Yaskawa INFORM job: R1_72,2(0,0)R2.JBI

/JOB
//NAME R1_72,2(0,0)R2
///FOLDERNAME KRIS-SCIANA
//POS
///NPOS 57,57,0,3,0,0
///TOOL 0
///POSTYPE PULSE
///PULSE
C00000=120729,38464,-23607,67702,92694,37114
C00001=130813,19897,-28859,40674,87554,31415
C00002=125083,56704,30738,54224,74995,24956
C00003=126358,57000,31561,53980,74051,25086
C00004=124721,62288,44734,63185,73473,22335
C00005=124721,62512,45919,63338,73183,22075
C00006=124721,62288,44734,63185,73473,22335
C00007=125305,62416,44881,63099,73087,22421
C00008=124721,62288,44734,63185,73473,22335
C00009=120729,38464,-23607,67702,92694,37114
C00010=120728,81583,44137,67576,84483,28591
C00011=120728,81849,43244,67535,84761,28882
C00012=120728,81417,45180,67625,84187,28282
C00013=120728,81508,44709,67602,84324,28425
C00014=119180,81573,44789,67929,85318,28213
C00015=119180,81465,45362,67951,85156,28039
C00016=120171,81410,45292,67747,84521,28174
C00017=118840,81840,43784,67968,85844,28487
C00018=118840,81840,43784,67968,85844,28487
C00019=120728,81522,44639,67599,84344,28446
C00020=120728,81598,44155,67576,84481,28590
C00021=121739,82345,42246,50477,71891,30249
C00022=121737,83430,44678,50707,71287,29904
C00023=121727,86673,48704,50914,70767,29601
C00024=120728,82318,42212,50838,72434,30029
C00025=120728,82318,42212,50838,72434,30029
C00026=120728,83470,39162,50303,74040,30931
C00027=120731,108704,30437,520,103146,-53106
C00028=120730,95364,30685,507,96140,-53135
C00029=120729,92856,31465,505,94371,-53142
C00030=120882,90601,30856,459,93584,-53097
C00031=120076,91948,31897,698,93643,-53342
C00032=120729,92386,31163,506,94315,-53143
C00033=120916,97871,39788,450,91825,-53093
C00034=121066,129805,79437,461,95361,-53027
C00035=121134,131914,82339,451,94657,-53008
C00036=120821,132587,79324,499,96860,-53101
C00037=120730,97149,30254,16854,109142,-86058
C00038=94374,59905,-24624,-6692,95808,-73268
C00039=94859,43835,-17383,-4554,74801,-71238
C00040=94859,41415,-16000,-4599,72712,-71159
C00041=88285,47191,-10324,7479,76594,-70277
C00042=94590,38531,-17304,-4457,72022,-71215
C00043=94826,41033,-16151,-4582,72608,-71165
C00044=88838,46898,-10539,7187,76531,-70115
C00045=90938,44895,-12618,6065,76637,-69484
C00046=101911,56037,-3137,-16386,82833,-70668
C00047=102467,62438,3678,-16668,82058,-70394
C00048=102039,71942,670,-16368,88461,-71374
C00049=120729,38464,-23607,67702,92694,37114
C00050=126358,57000,31561,53980,74051,25086
C00051=127340,53488,29402,53838,73202,25111
C00052=126498,52546,32838,59465,71466,23946
C00053=126411,61917,43233,59752,70711,23276
C00054=125699,61499,41475,59654,71606,23502
C00055=127963,-13691,-44237,56024,78067,29543
C00056=48492,61943,-11432,-541,72797,-1948
BC00000=247969,581384,1069855
BC00001=247969,581384,399097
BC00002=247969,581384,399097
BC00003=247969,581384,399097
BC00004=247969,581384,399097
BC00005=247969,581384,399097
BC00006=247969,581384,399097
BC00007=247969,581384,399097
BC00008=247969,581384,399097
BC00009=247969,581384,1069855
BC00010=247969,581384,1069855
BC00011=234047,579018,1046735
BC00012=234047,579018,1046735
BC00013=234047,579018,1046735
BC00014=234047,579018,1046735
BC00015=234047,579018,1046735
BC00016=234047,579018,1046735
BC00017=234047,579018,1046735
BC00018=234047,579018,1046735
BC00019=234047,579018,1046735
BC00020=240166,577093,1047559
BC00021=204016,615205,1075175
BC00022=204016,615205,1075175
BC00023=204016,615205,1075175
BC00024=204016,615205,1075175
BC00025=204016,615205,1075175
BC00026=222293,612873,1075175
BC00027=148834,597684,1075175
BC00028=148876,597689,1075175
BC00029=146152,596166,1075175
BC00030=145063,595557,1075175
BC00031=145063,595557,1075175
BC00032=145063,595557,1075175
BC00033=145063,595557,1075175
BC00034=145063,595557,1075175
BC00035=145063,595557,1075175
BC00036=145063,595557,1075175
BC00037=163962,558925,1075175
BC00038=16042,566310,1075175
BC00039=16207,572657,1075175
BC00040=16871,569169,1075175
BC00041=17137,567774,1075175
BC00042=17137,567774,1075175
BC00043=17137,567774,1075175
BC00044=17137,567774,1075175
BC00045=17137,567774,1075175
BC00046=17137,567774,1075175
BC00047=17137,567774,1075175
BC00048=17137,567774,1075175
BC00049=247969,581384,1069855
BC00050=247969,581384,399097
BC00051=247969,581384,399097
BC00052=247969,581384,399097
BC00053=247969,581384,399097
BC00054=247969,581384,399097
BC00055=247969,581384,399097
BC00056=49225,622868,1075175
///POSTYPE BASE
///RECTAN
///RCONF 0,0,0,0,1,0,0,0,0,0,0,0,0,0,0,0,0,0,0,0,0,0,0,0
P00006=2.006,1.622,-0.565,0.0000,0.0000,0.0000
P00021=0.073,2.058,-0.109,0.0000,0.0000,0.0000
///RCONF 0,0,0,0,0,0,0,0,0,0,0,0,0,0,0,0,0,0,0,0,0,0,0,0
P00030=-0.014,-0.768,0.131,0.0000,0.0000,0.0000
//INST
///DATE 2025/03/04 15:05
///ATTR SC,RW
///GROUP1 RB1,BS1
NOP
'R2_72.2(0,0)
'Path S1184
SFTOF
MOVJ C00000 BC00000 VJ=100.00
MOVJ C00001 BC00001 VJ=100.00
MOVJ C00002 BC00002 VJ=100.00
MOVL C00003 BC00003 V=166.7
MOVL C00004 BC00004 V=100.0
REFP 3 C00005 BC00005
CALL JOB:SEARCH-R1
SET P030 P006
SFTON P030
MOVL C00006 BC00006 V=100.0
REFP 3 C00007 BC00007
CALL JOB:SEARCH-R1
SET P030 P006
SFTON P030
MOVL C00008 BC00008 V=100.0
SFTOF
MOVJ C00009 BC00009 VJ=100.00
MOVJ C00010 BC00010 VJ=100.00
MOVL C00011 BC00011 V=100.0
REFP 3 C00012 BC00012
CALL JOB:SEARCH-R1
SET P021 P006
SFTON P021
MOVL C00013 BC00013 V=100.0
MOVL C00014 BC00014 V=100.0
MOVL C00015 BC00015 V=60.0
REFP 3 C00016 BC00016
CALL JOB:SEARCH-R1
SET P021 P006
SFTON P021
MOVL C00017 BC00017 V=60.0
MOVL C00018 BC00018 V=100.0
MOVL C00019 BC00019 V=60.0
MOVL C00020 BC00020 V=100.0
MOVL C00021 BC00021 V=100.0
MOVL C00022 BC00022 V=60.0
REFP 3 C00023 BC00023
CALL JOB:SEARCH-R1
SET P021 P006
SFTON P021
MOVL C00024 BC00024 V=60.0
MOVL C00025 BC00025 V=100.0
MOVL C00026 BC00026 V=100.0
'Path W1186
SFTOF
SFTON P021
MOVJ C00027 BC00027 VJ=100.00
MOVJ C00028 BC00028 VJ=100.00
MOVL C00029 BC00029 V=100.0
CALL JOB:COFNIJ_DRUT
MOVL C00030 BC00030 V=100.0 PL=0
REFP 1 C00031 BC00031
REFP 2 C00032 BC00032
MACRO1 MJ#(0) ARGF6
ARCON
MOVL C00033 BC00033 V=10.8
MOVL C00034 BC00034 V=10.8
MOVL C00035 BC00035 V=10.0
ARCOF
MOVL C00036 BC00036 V=100.0
MOVL C00037 BC00037 V=100.0
SFTOF
'Path W1188
SFTOF
SFTON P021
MOVJ C00038 BC00038 VJ=100.00
MOVJ C00039 BC00039 VJ=100.00
MOVJ C00040 BC00040 VJ=100.00
MOVL C00041 BC00041 V=100.0 PL=0
REFP 1 C00042 BC00042
REFP 2 C00043 BC00043
MACRO1 MJ#(0) ARGF6
ARCON
MOVL C00044 BC00044 V=8.3
MOVL C00045 BC00045 V=8.3
MOVL C00046 BC00046 V=8.3
MOVL C00047 BC00047 V=8.3
ARCOF
MOVL C00048 BC00048 V=100.0
SFTOF
MOVJ C00049 BC00049 VJ=100.00
MOVL C00050 BC00050 V=400.0
SFTON P030
MOVL C00051 BC00051 V=166.7
MOVL C00052 BC00052 V=100.0 PL=0
MACRO1 MJ#(0) ARGF7
ARCON
MOVL C00053 BC00053 V=9.2
ARCOF
MOVL C00054 BC00054 V=166.7
SFTOF
MOVJ C00055 BC00055 VJ=100.00
MOVJ C00056 BC00056 VJ=100.00
SFTOF
END
